GLOBALCONSTANTS LO (* Global constants Modules with low IO density *)
  (* Standard: 61499-1; Description: Copyright (c) 2024 HR Agrartechnik GmbH This program and the accompanying materials are made available under the terms of the Eclipse Public License 2.0 which is available at https://www.eclipse.org/legal/epl-2.0/ SPDX-License-Identifier: EPL-2.0 *)
  (* Version 1.0, 2024-01-25, Franz Höpfinger, HR Agrartechnik GmbH *)
  PACKAGE DataPanel::io::LO::const;
  VAR_GLOBAL CONSTANT
    LO_00 : USINT := 217;
    LO_01 : USINT := 218;
    LO_02 : USINT := 219;
    LO_03 : USINT := 220;
    LO_04 : USINT := 221;
    LO_05 : USINT := 222;
    LO_06 : USINT := 223;
    LO_07 : USINT := 224;
  END_VAR
END_GLOBALCONSTANTS
